// TIA Portal V15.1 export
// export: Created 2024-06-21T08:40:58.1290505Z, ExportSetting WithDefaults, DisplayName Totally Integrated Automation Portal, DisplayVersion V15.1 Update 5, DisplayName TIA Portal Openness, DisplayVersion V15.1 Update 5, DisplayName SINAMICS Startdrive Advanced, DisplayVersion V15.1, DisplayName G130, G150, S120, S150, SINAMICS MV, S210, DisplayVersion V15.1, DisplayName G110M, G120, G120C, G120D, G120P, DisplayVersion V15.1, DisplayName STEP 7 Professional, DisplayVersion V15.1 Update 5, DisplayName STEP 7 Safety, DisplayVersion V15.1, DisplayName WinCC Professional, DisplayVersion V15.1 Update 5, DisplayName SIMATIC Visualization Architect, DisplayVersion V15.1
FUNCTION_BLOCK "LETAFuseCPC20PN"   // FB1406, FBD
TITLE = LETAFuseCPC20PN
{ S7_Optimized_Access := 'TRUE' }
AUTHOR : VCC
FAMILY : AlarmHnd
VERSION : 0.1
// stored: AutoNumber false, IsIECCheckEnabled false, IsRetainMemResEnabled false, MemoryReserve 100, SetENOAutomatically False, UDAEnableTagReadback false
   VAR_INPUT
      I_NewShift { ExternalAccessible := 'False'; ExternalVisible := 'False'; ExternalWritable := 'False'} : Bool;   // NewShift / Morning shift
      I_EnableAlarm { ExternalAccessible := 'False'; ExternalVisible := 'False'; ExternalWritable := 'False'} : Bool := TRUE;   // Enable Alarm from upper level
      C_HWInput { ExternalAccessible := 'False'; ExternalVisible := 'False'; ExternalWritable := 'False'} : HW_IO;   // Slot ID from CPC20PN
      C_Block1_TotalCurrent { ExternalAccessible := 'False'; ExternalVisible := 'False'; ExternalWritable := 'False'} : HW_IO;   // Base Module Slot ID Total Current, 0=not in use.
      C_Block1_StatusControl { ExternalAccessible := 'False'; ExternalVisible := 'False'; ExternalWritable := 'False'} : HW_IO;   // Base Module Slot ID Status / Control, 0=not in use.
      "C_Block1_MeasurementU/I" { ExternalAccessible := 'False'; ExternalVisible := 'False'; ExternalWritable := 'False'} : HW_IO;   // Base Module Slot ID Measurement UI, 0=not in use.
      C_Block2_TotalCurrent { ExternalAccessible := 'False'; ExternalVisible := 'False'; ExternalWritable := 'False'} : HW_IO;   // Extension Module Slot ID Total Current, 0=not in use.
      C_Block2_StatusControl { ExternalAccessible := 'False'; ExternalVisible := 'False'; ExternalWritable := 'False'} : HW_IO;   // Extension Module Slot ID Status / Control, 0=not in use.
      "C_Block2_MeasurementU/I" { ExternalAccessible := 'False'; ExternalVisible := 'False'; ExternalWritable := 'False'} : HW_IO;   // Extension Module Slot ID Measurement UI, 0=not in use.
      C_Config { ExternalAccessible := 'False'; ExternalVisible := 'False'; ExternalWritable := 'False'} : "ETAFuseCPC20PNConfig";   // Config
   END_VAR
   VAR_OUTPUT
      O_AlarmABCondition { ExternalAccessible := 'False'; ExternalVisible := 'False'; ExternalWritable := 'False'} : Bool;   // Alarm AB Condition
      O_AlarmA { ExternalAccessible := 'False'; ExternalVisible := 'False'; ExternalWritable := 'False'} : Bool;   // Alarm A
      O_AlarmB { ExternalAccessible := 'False'; ExternalVisible := 'False'; ExternalWritable := 'False'} : Bool;   // Alarm B
      O_AlarmC { ExternalAccessible := 'False'; ExternalVisible := 'False'; ExternalWritable := 'False'} : Bool;   // Alarm C
      O_AlarmD { ExternalAccessible := 'False'; ExternalVisible := 'False'; ExternalWritable := 'False'} : Bool;   // Alarm D
      H_AlarmDWord { ExternalAccessible := 'False'; ExternalVisible := 'False'; ExternalWritable := 'False'} : DWord;   // HMI Animation
   END_VAR
   VAR_IN_OUT
      IO_ETAFuseData : "ETAFuseData";   // ETA fuse status
      H_HMI : "H_HMI";   // Animation
      H_ETAFuseCPC20PN : "H_ETAFuseCPC20PN";   // Animation
   END_VAR
   VAR
      AC_StatusCPC20_Bit0 { ExternalAccessible := 'False'; ExternalVisible := 'False'; ExternalWritable := 'False'} : Bool;   // No configuration data available
      AC_StatusCPC20_Bit1 { ExternalAccessible := 'False'; ExternalVisible := 'False'; ExternalWritable := 'False'} : Bool;   // Invalid configuration data
      AC_StatusCPC20_Bit4 { ExternalAccessible := 'False'; ExternalVisible := 'False'; ExternalWritable := 'False'} : Bool;   // Command buffer overflow
      AC_StatusCPC20_Bit7 { ExternalAccessible := 'False'; ExternalVisible := 'False'; ExternalWritable := 'False'} : Bool;   // No communication with at least one PWR board
      AC_StatusCPC20_Bit9 { ExternalAccessible := 'False'; ExternalVisible := 'False'; ExternalWritable := 'False'} : Bool;   // CPC tempory error
      AC_StatusCPC20_Bit10 { ExternalAccessible := 'False'; ExternalVisible := 'False'; ExternalWritable := 'False'} : Bool;   // CPC hardware error
      AC_ReadNomCurr { ExternalAccessible := 'False'; ExternalVisible := 'False'; ExternalWritable := 'False'} : Bool;   // Overtime Reading of nominal current
      AlarmABCondition { ExternalAccessible := 'False'; ExternalVisible := 'False'; ExternalWritable := 'False'} : Bool;   // Alarm AB Condition
      AlarmA { ExternalAccessible := 'False'; ExternalVisible := 'False'; ExternalWritable := 'False'} : Bool;   // Alarm A
      AlarmB { ExternalAccessible := 'False'; ExternalVisible := 'False'; ExternalWritable := 'False'} : Bool;   // Alarm B
      AlarmC { ExternalAccessible := 'False'; ExternalVisible := 'False'; ExternalWritable := 'False'} : Bool;   // Alarm C
      AlarmD { ExternalAccessible := 'False'; ExternalVisible := 'False'; ExternalWritable := 'False'} : Bool;   // Alarm D
      ReadNominalCurrentActive { ExternalAccessible := 'False'; ExternalVisible := 'False'; ExternalWritable := 'False'} : Bool;   // Reading of nominal current is active
      EnableAlarm { ExternalAccessible := 'False'; ExternalVisible := 'False'; ExternalWritable := 'False'} : Bool;   // Enable Alarm from upper level
   END_VAR
   VAR RETAIN
      H_ReadNomCurr { ExternalAccessible := 'False'; ExternalVisible := 'False'; ExternalWritable := 'False'} : Bool;   // HMI Command - Read nominal current
      H_CancelReadNomCurr { ExternalAccessible := 'False'; ExternalVisible := 'False'; ExternalWritable := 'False'} : Bool;   // HMI Command - Cancel Read nominal current
   END_VAR
   VAR
      H_UpChannel { ExternalAccessible := 'False'; ExternalVisible := 'False'; ExternalWritable := 'False'} : Bool;   // HMI Command - UP channel selection
      H_DownChannel { ExternalAccessible := 'False'; ExternalVisible := 'False'; ExternalWritable := 'False'} : Bool;   // HMI Command - DOWN channel selection
      H_SwitchON { ExternalAccessible := 'False'; ExternalVisible := 'False'; ExternalWritable := 'False'} : Bool;   // HMICmd / HMI Command - Switch On
      H_SwitchOFF { ExternalAccessible := 'False'; ExternalVisible := 'False'; ExternalWritable := 'False'} : Bool;   // HMICmd / HMI Command - Switch Off
      H_Transfer { ExternalAccessible := 'False'; ExternalVisible := 'False'; ExternalWritable := 'False'} : Bool;   // HMICmd / HMI Command - Transfer
      H_Reset { ExternalAccessible := 'False'; ExternalVisible := 'False'; ExternalWritable := 'False'} : Bool;   // HMICmd / HMI Command - Reset
      _ETAFuseCPC20PNSub { ExternalAccessible := 'False'; ExternalVisible := 'False'; ExternalWritable := 'False'} : "LETAFuseCPC20PNSub";   // FB
   END_VAR
   VAR DB_SPECIFIC
      T_ResetControl { ExternalAccessible := 'False'; ExternalVisible := 'False'; ExternalWritable := 'False'} : TON_TIME;   // Timer
      T_EnableAlarm { ExternalAccessible := 'False'; ExternalVisible := 'False'; ExternalWritable := 'False'} : TON_TIME;   // Timer
   END_VAR
   VAR
      Edge { ExternalAccessible := 'False'; ExternalVisible := 'False'; ExternalWritable := 'False'} : Array[0..10] of Bool;   // Edge
   END_VAR
   VAR_TEMP   // added for the SCL form of the ladder/FBD networks
      _w1 : Bool;
      _w2 : Bool;
   END_VAR
BEGIN

REGION Network 1: **** 1 - Inputs **** Extract The Commands From HMI
   // Extract The Commands From HMI
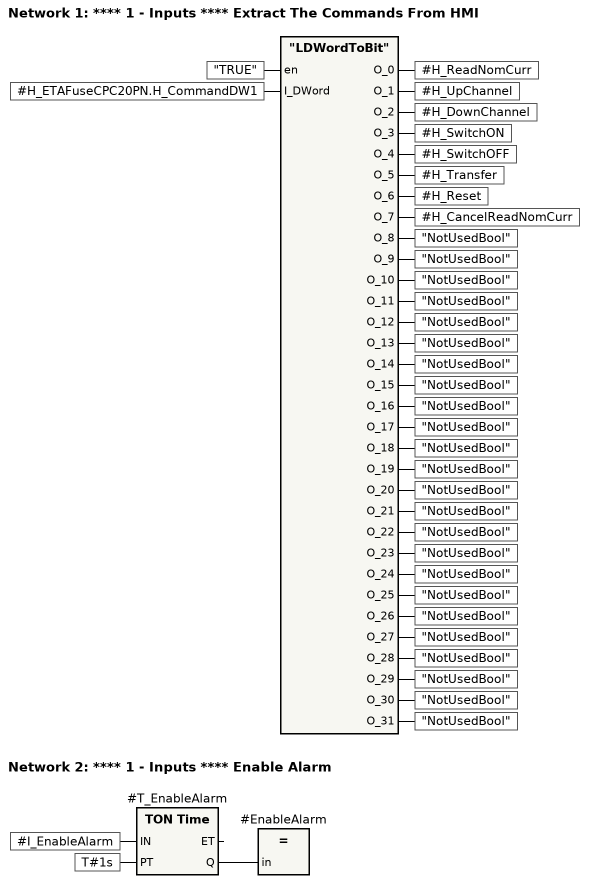
   IF "TRUE" THEN
       "LDWordToBit"(I_DWord := #H_ETAFuseCPC20PN.H_CommandDW1,
                     O_0 => #H_ReadNomCurr,
                     O_1 => #H_UpChannel,
                     O_2 => #H_DownChannel,
                     O_3 => #H_SwitchON,
                     O_4 => #H_SwitchOFF,
                     O_5 => #H_Transfer,
                     O_6 => #H_Reset,
                     O_7 => #H_CancelReadNomCurr,
                     O_8 => "NotUsedBool",
                     O_9 => "NotUsedBool",
                     O_10 => "NotUsedBool",
                     O_11 => "NotUsedBool",
                     O_12 => "NotUsedBool",
                     O_13 => "NotUsedBool",
                     O_14 => "NotUsedBool",
                     O_15 => "NotUsedBool",
                     O_16 => "NotUsedBool",
                     O_17 => "NotUsedBool",
                     O_18 => "NotUsedBool",
                     O_19 => "NotUsedBool",
                     O_20 => "NotUsedBool",
                     O_21 => "NotUsedBool",
                     O_22 => "NotUsedBool",
                     O_23 => "NotUsedBool",
                     O_24 => "NotUsedBool",
                     O_25 => "NotUsedBool",
                     O_26 => "NotUsedBool",
                     O_27 => "NotUsedBool",
                     O_28 => "NotUsedBool",
                     O_29 => "NotUsedBool",
                     O_30 => "NotUsedBool",
                     O_31 => "NotUsedBool");
   END_IF;
END_REGION

REGION Network 2: **** 1 - Inputs **** Enable Alarm
   #T_EnableAlarm(IN := #I_EnableAlarm, PT := T#1s);   // TON
   #EnableAlarm := #T_EnableAlarm.Q;
END_REGION

REGION Network 3: **** 4.3 - Machine status - Operator Selection **** Selected Channel
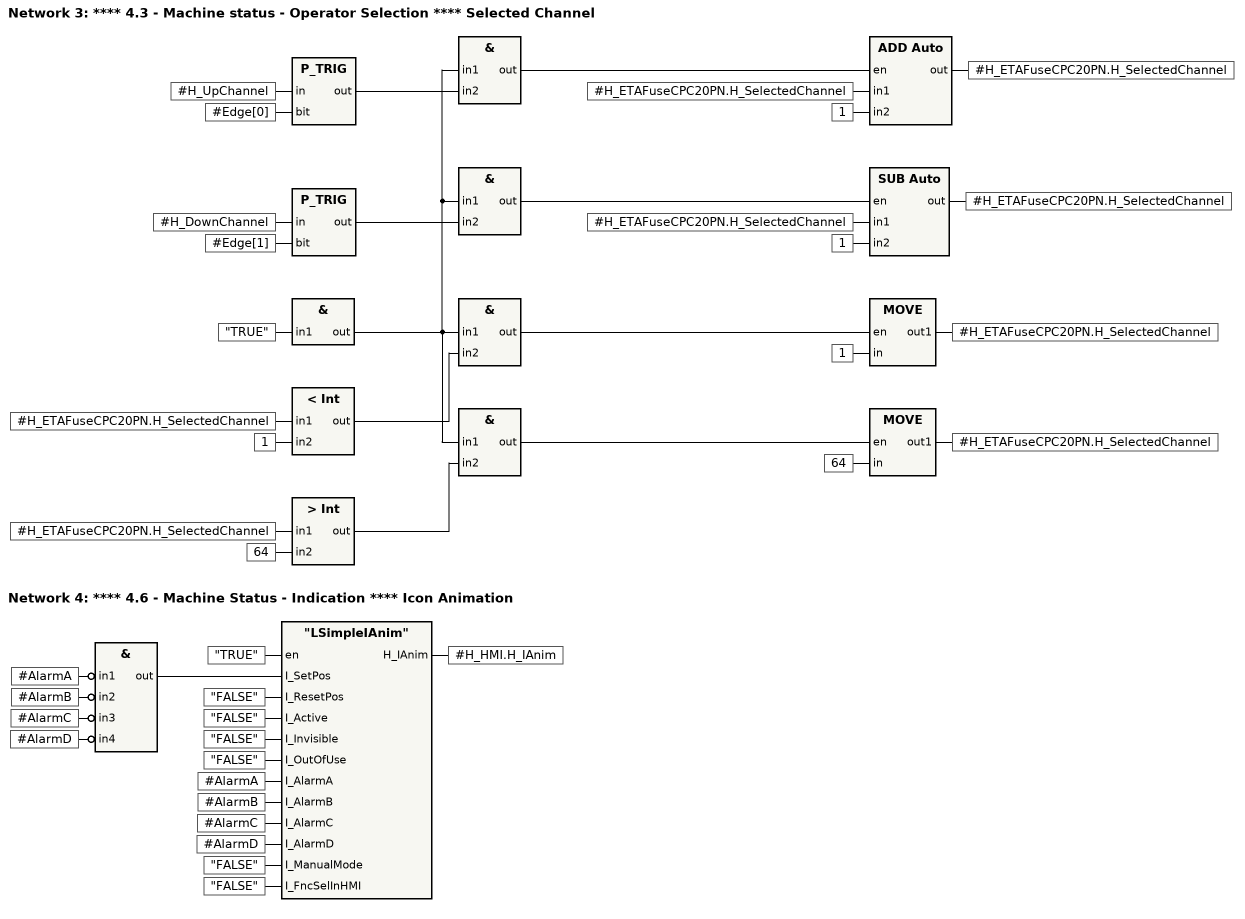
   #_w1 := #H_UpChannel AND NOT #Edge[0];   // rising edge
   #Edge[0] := #H_UpChannel;
   IF "TRUE" AND #_w1 THEN
       #H_ETAFuseCPC20PN.H_SelectedChannel := #H_ETAFuseCPC20PN.H_SelectedChannel + 1;
   END_IF;
   #_w2 := #H_DownChannel AND NOT #Edge[1];   // rising edge
   #Edge[1] := #H_DownChannel;
   IF "TRUE" AND #_w2 THEN
       #H_ETAFuseCPC20PN.H_SelectedChannel := #H_ETAFuseCPC20PN.H_SelectedChannel - 1;
   END_IF;
   IF "TRUE" AND (#H_ETAFuseCPC20PN.H_SelectedChannel < 1) THEN
       #H_ETAFuseCPC20PN.H_SelectedChannel := 1;
   END_IF;
   IF "TRUE" AND (#H_ETAFuseCPC20PN.H_SelectedChannel > 64) THEN
       #H_ETAFuseCPC20PN.H_SelectedChannel := 64;
   END_IF;
END_REGION

REGION Network 4: **** 4.6 - Machine Status - Indication **** Icon Animation
   // Icon Animation
   IF "TRUE" THEN
       "LSimpleIAnim"(I_SetPos := NOT #AlarmA AND NOT #AlarmB AND NOT #AlarmC AND NOT #AlarmD,
                      I_ResetPos := "FALSE",
                      I_Active := "FALSE",
                      I_Invisible := "FALSE",
                      I_OutOfUse := "FALSE",
                      I_AlarmA := #AlarmA,
                      I_AlarmB := #AlarmB,
                      I_AlarmC := #AlarmC,
                      I_AlarmD := #AlarmD,
                      I_ManualMode := "FALSE",
                      I_FncSelInHMI := "FALSE",
                      H_IAnim => #H_HMI.H_IAnim);
   END_IF;
END_REGION

REGION Network 5: **** 4.6 - Machine Status - Indication **** Animation
   // Animation
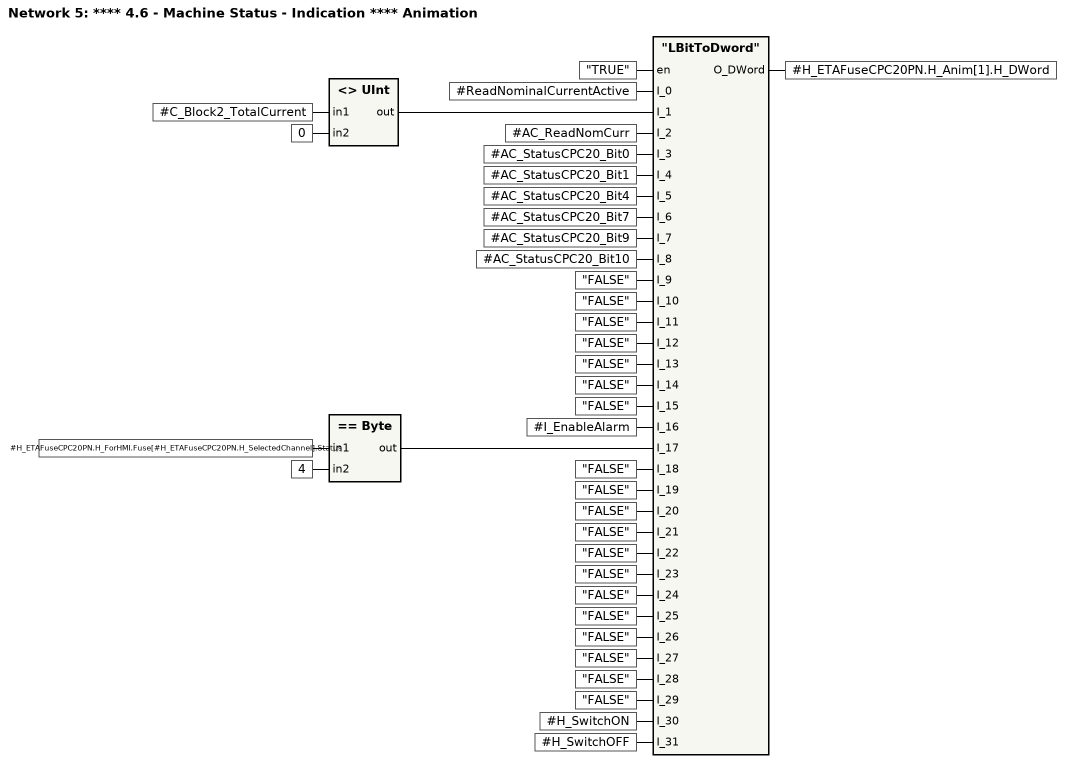
   IF "TRUE" THEN
       "LBitToDword"(I_0 := #ReadNominalCurrentActive,
                     I_1 := #C_Block2_TotalCurrent <> 0,
                     I_2 := #AC_ReadNomCurr,
                     I_3 := #AC_StatusCPC20_Bit0,
                     I_4 := #AC_StatusCPC20_Bit1,
                     I_5 := #AC_StatusCPC20_Bit4,
                     I_6 := #AC_StatusCPC20_Bit7,
                     I_7 := #AC_StatusCPC20_Bit9,
                     I_8 := #AC_StatusCPC20_Bit10,
                     I_9 := "FALSE",
                     I_10 := "FALSE",
                     I_11 := "FALSE",
                     I_12 := "FALSE",
                     I_13 := "FALSE",
                     I_14 := "FALSE",
                     I_15 := "FALSE",
                     I_16 := #I_EnableAlarm,
                     I_17 := #H_ETAFuseCPC20PN.H_ForHMI.Fuse[#H_ETAFuseCPC20PN.H_SelectedChannel].Status = 4,
                     I_18 := "FALSE",
                     I_19 := "FALSE",
                     I_20 := "FALSE",
                     I_21 := "FALSE",
                     I_22 := "FALSE",
                     I_23 := "FALSE",
                     I_24 := "FALSE",
                     I_25 := "FALSE",
                     I_26 := "FALSE",
                     I_27 := "FALSE",
                     I_28 := "FALSE",
                     I_29 := "FALSE",
                     I_30 := #H_SwitchON,
                     I_31 := #H_SwitchOFF,
                     O_DWord => #H_ETAFuseCPC20PN.H_Anim[1].H_DWord);
   END_IF;
END_REGION

REGION Network 6: **** 4.6 - Machine Status - Indication **** Animation
   // Animation
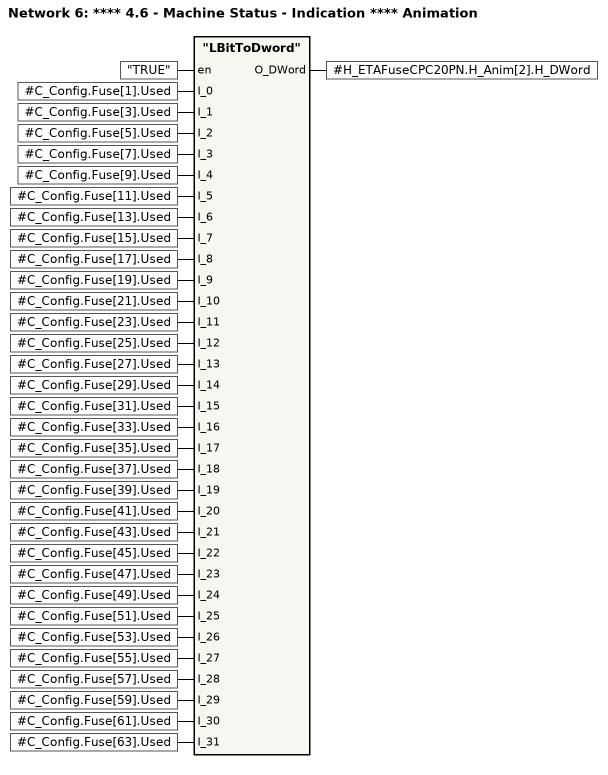
   IF "TRUE" THEN
       "LBitToDword"(I_0 := #C_Config.Fuse[1].Used,
                     I_1 := #C_Config.Fuse[3].Used,
                     I_2 := #C_Config.Fuse[5].Used,
                     I_3 := #C_Config.Fuse[7].Used,
                     I_4 := #C_Config.Fuse[9].Used,
                     I_5 := #C_Config.Fuse[11].Used,
                     I_6 := #C_Config.Fuse[13].Used,
                     I_7 := #C_Config.Fuse[15].Used,
                     I_8 := #C_Config.Fuse[17].Used,
                     I_9 := #C_Config.Fuse[19].Used,
                     I_10 := #C_Config.Fuse[21].Used,
                     I_11 := #C_Config.Fuse[23].Used,
                     I_12 := #C_Config.Fuse[25].Used,
                     I_13 := #C_Config.Fuse[27].Used,
                     I_14 := #C_Config.Fuse[29].Used,
                     I_15 := #C_Config.Fuse[31].Used,
                     I_16 := #C_Config.Fuse[33].Used,
                     I_17 := #C_Config.Fuse[35].Used,
                     I_18 := #C_Config.Fuse[37].Used,
                     I_19 := #C_Config.Fuse[39].Used,
                     I_20 := #C_Config.Fuse[41].Used,
                     I_21 := #C_Config.Fuse[43].Used,
                     I_22 := #C_Config.Fuse[45].Used,
                     I_23 := #C_Config.Fuse[47].Used,
                     I_24 := #C_Config.Fuse[49].Used,
                     I_25 := #C_Config.Fuse[51].Used,
                     I_26 := #C_Config.Fuse[53].Used,
                     I_27 := #C_Config.Fuse[55].Used,
                     I_28 := #C_Config.Fuse[57].Used,
                     I_29 := #C_Config.Fuse[59].Used,
                     I_30 := #C_Config.Fuse[61].Used,
                     I_31 := #C_Config.Fuse[63].Used,
                     O_DWord => #H_ETAFuseCPC20PN.H_Anim[2].H_DWord);
   END_IF;
END_REGION

REGION Network 7: **** 4.6 - Machine Status - Indication **** Animation
   // Animation
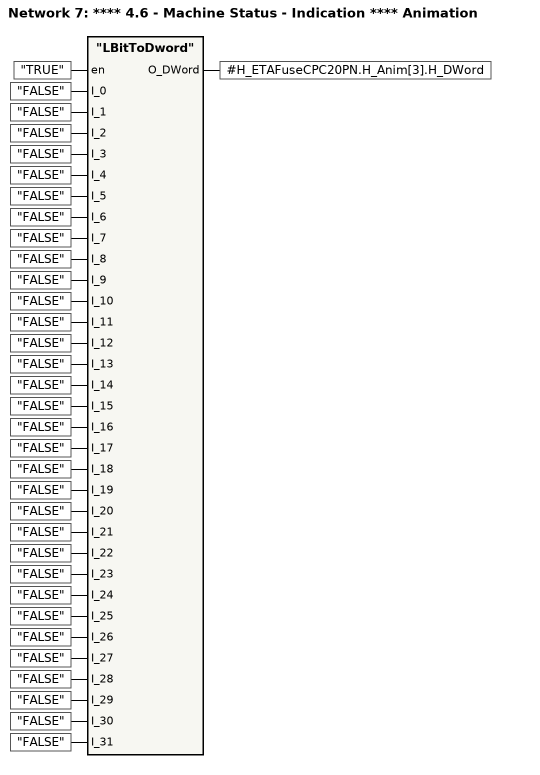
   IF "TRUE" THEN
       "LBitToDword"(I_0 := "FALSE",
                     I_1 := "FALSE",
                     I_2 := "FALSE",
                     I_3 := "FALSE",
                     I_4 := "FALSE",
                     I_5 := "FALSE",
                     I_6 := "FALSE",
                     I_7 := "FALSE",
                     I_8 := "FALSE",
                     I_9 := "FALSE",
                     I_10 := "FALSE",
                     I_11 := "FALSE",
                     I_12 := "FALSE",
                     I_13 := "FALSE",
                     I_14 := "FALSE",
                     I_15 := "FALSE",
                     I_16 := "FALSE",
                     I_17 := "FALSE",
                     I_18 := "FALSE",
                     I_19 := "FALSE",
                     I_20 := "FALSE",
                     I_21 := "FALSE",
                     I_22 := "FALSE",
                     I_23 := "FALSE",
                     I_24 := "FALSE",
                     I_25 := "FALSE",
                     I_26 := "FALSE",
                     I_27 := "FALSE",
                     I_28 := "FALSE",
                     I_29 := "FALSE",
                     I_30 := "FALSE",
                     I_31 := "FALSE",
                     O_DWord => #H_ETAFuseCPC20PN.H_Anim[3].H_DWord);
   END_IF;
END_REGION

REGION Network 8: **** 4.6 - Machine Status - Indication **** Animation
   // Animation
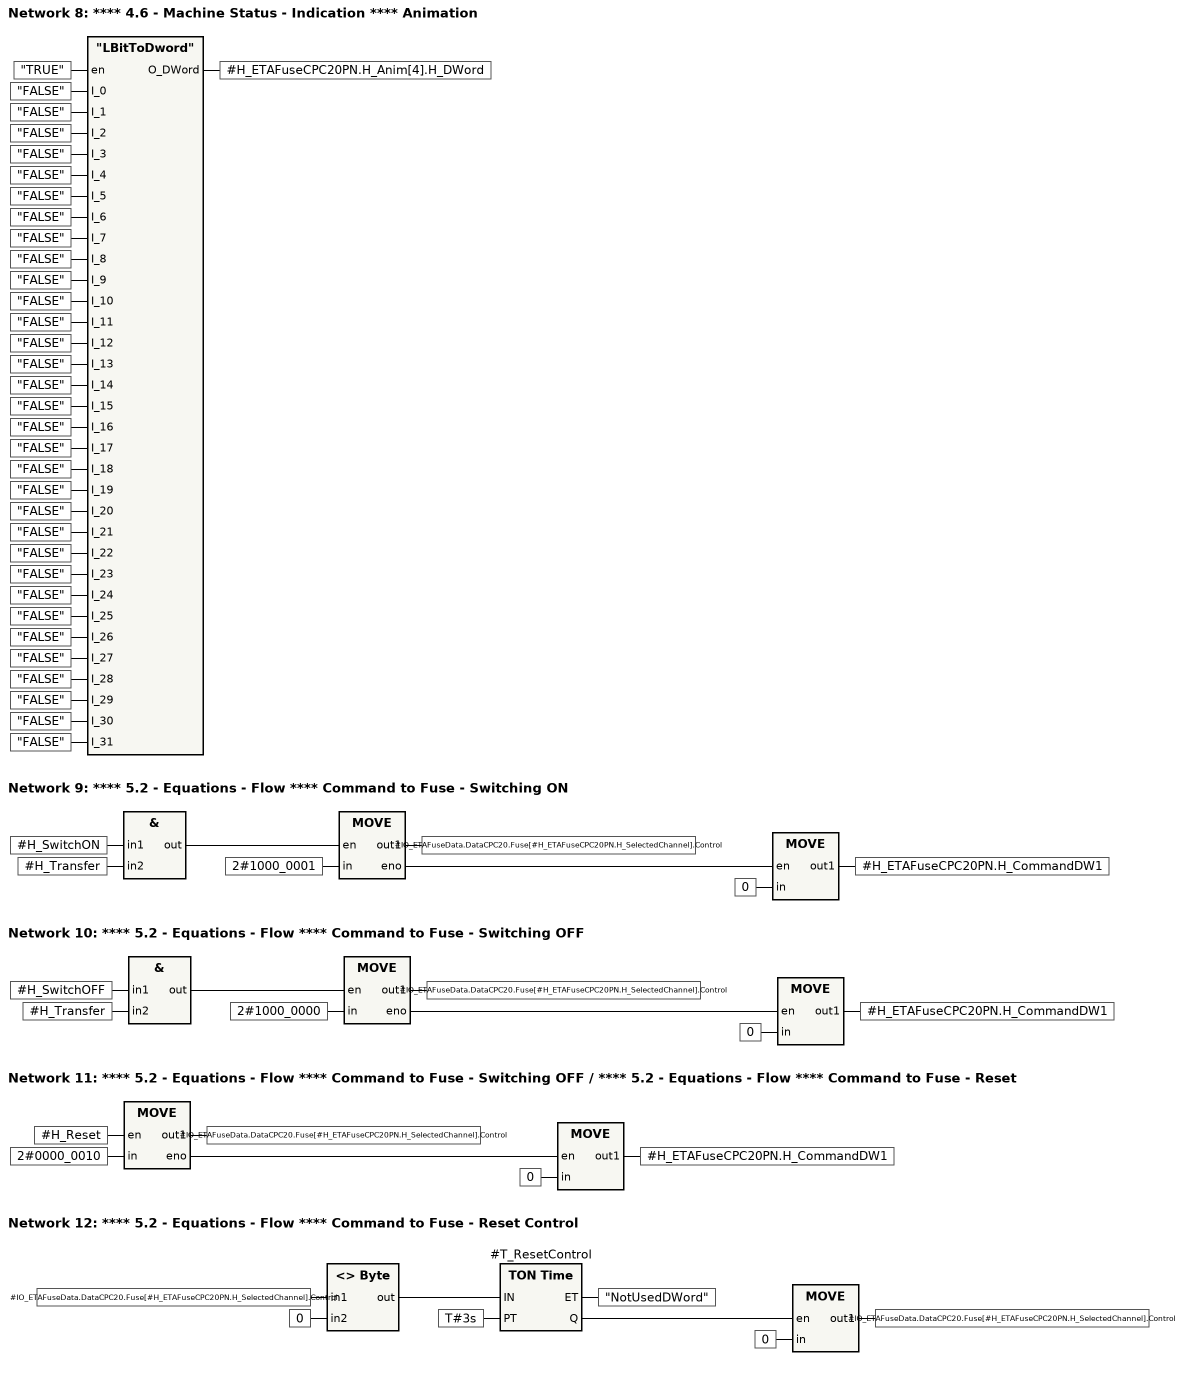
   IF "TRUE" THEN
       "LBitToDword"(I_0 := "FALSE",
                     I_1 := "FALSE",
                     I_2 := "FALSE",
                     I_3 := "FALSE",
                     I_4 := "FALSE",
                     I_5 := "FALSE",
                     I_6 := "FALSE",
                     I_7 := "FALSE",
                     I_8 := "FALSE",
                     I_9 := "FALSE",
                     I_10 := "FALSE",
                     I_11 := "FALSE",
                     I_12 := "FALSE",
                     I_13 := "FALSE",
                     I_14 := "FALSE",
                     I_15 := "FALSE",
                     I_16 := "FALSE",
                     I_17 := "FALSE",
                     I_18 := "FALSE",
                     I_19 := "FALSE",
                     I_20 := "FALSE",
                     I_21 := "FALSE",
                     I_22 := "FALSE",
                     I_23 := "FALSE",
                     I_24 := "FALSE",
                     I_25 := "FALSE",
                     I_26 := "FALSE",
                     I_27 := "FALSE",
                     I_28 := "FALSE",
                     I_29 := "FALSE",
                     I_30 := "FALSE",
                     I_31 := "FALSE",
                     O_DWord => #H_ETAFuseCPC20PN.H_Anim[4].H_DWord);
   END_IF;
END_REGION

REGION Network 9: **** 5.2 - Equations - Flow **** Command to Fuse - Switching ON
   // Switching ON
   // ENO of a box is taken as its EN; it also drops when the box reports an error
   IF #H_SwitchON AND #H_Transfer THEN
       #IO_ETAFuseData.DataCPC20.Fuse[#H_ETAFuseCPC20PN.H_SelectedChannel].Control := 2#1000_0001;
       #H_ETAFuseCPC20PN.H_CommandDW1 := 0;
   END_IF;
END_REGION

REGION Network 10: **** 5.2 - Equations - Flow **** Command to Fuse - Switching OFF
   // Switching OFF
   // ENO of a box is taken as its EN; it also drops when the box reports an error
   IF #H_SwitchOFF AND #H_Transfer THEN
       #IO_ETAFuseData.DataCPC20.Fuse[#H_ETAFuseCPC20PN.H_SelectedChannel].Control := 2#1000_0000;
       #H_ETAFuseCPC20PN.H_CommandDW1 := 0;
   END_IF;
END_REGION

REGION Network 11: **** 5.2 - Equations - Flow **** Command to Fuse - Switching OFF / **** 5.2 - Equations - Flow **** Command to Fuse - Reset
   // Switching OFF / Reset
   // ENO of a box is taken as its EN; it also drops when the box reports an error
   IF #H_Reset THEN
       #IO_ETAFuseData.DataCPC20.Fuse[#H_ETAFuseCPC20PN.H_SelectedChannel].Control := 2#0000_0010;
       #H_ETAFuseCPC20PN.H_CommandDW1 := 0;
   END_IF;
END_REGION

REGION Network 12: **** 5.2 - Equations - Flow **** Command to Fuse - Reset Control
   #T_ResetControl(IN := #IO_ETAFuseData.DataCPC20.Fuse[#H_ETAFuseCPC20PN.H_SelectedChannel].Control <> 0,   // TON
                   PT := T#3s,
                   ET => "NotUsedDWord");
   IF #T_ResetControl.Q THEN
       #IO_ETAFuseData.DataCPC20.Fuse[#H_ETAFuseCPC20PN.H_SelectedChannel].Control := 0;
   END_IF;
END_REGION

REGION Network 13: **** 7.1 - Submodule - Non-Machine **** ETA CPC20 PN
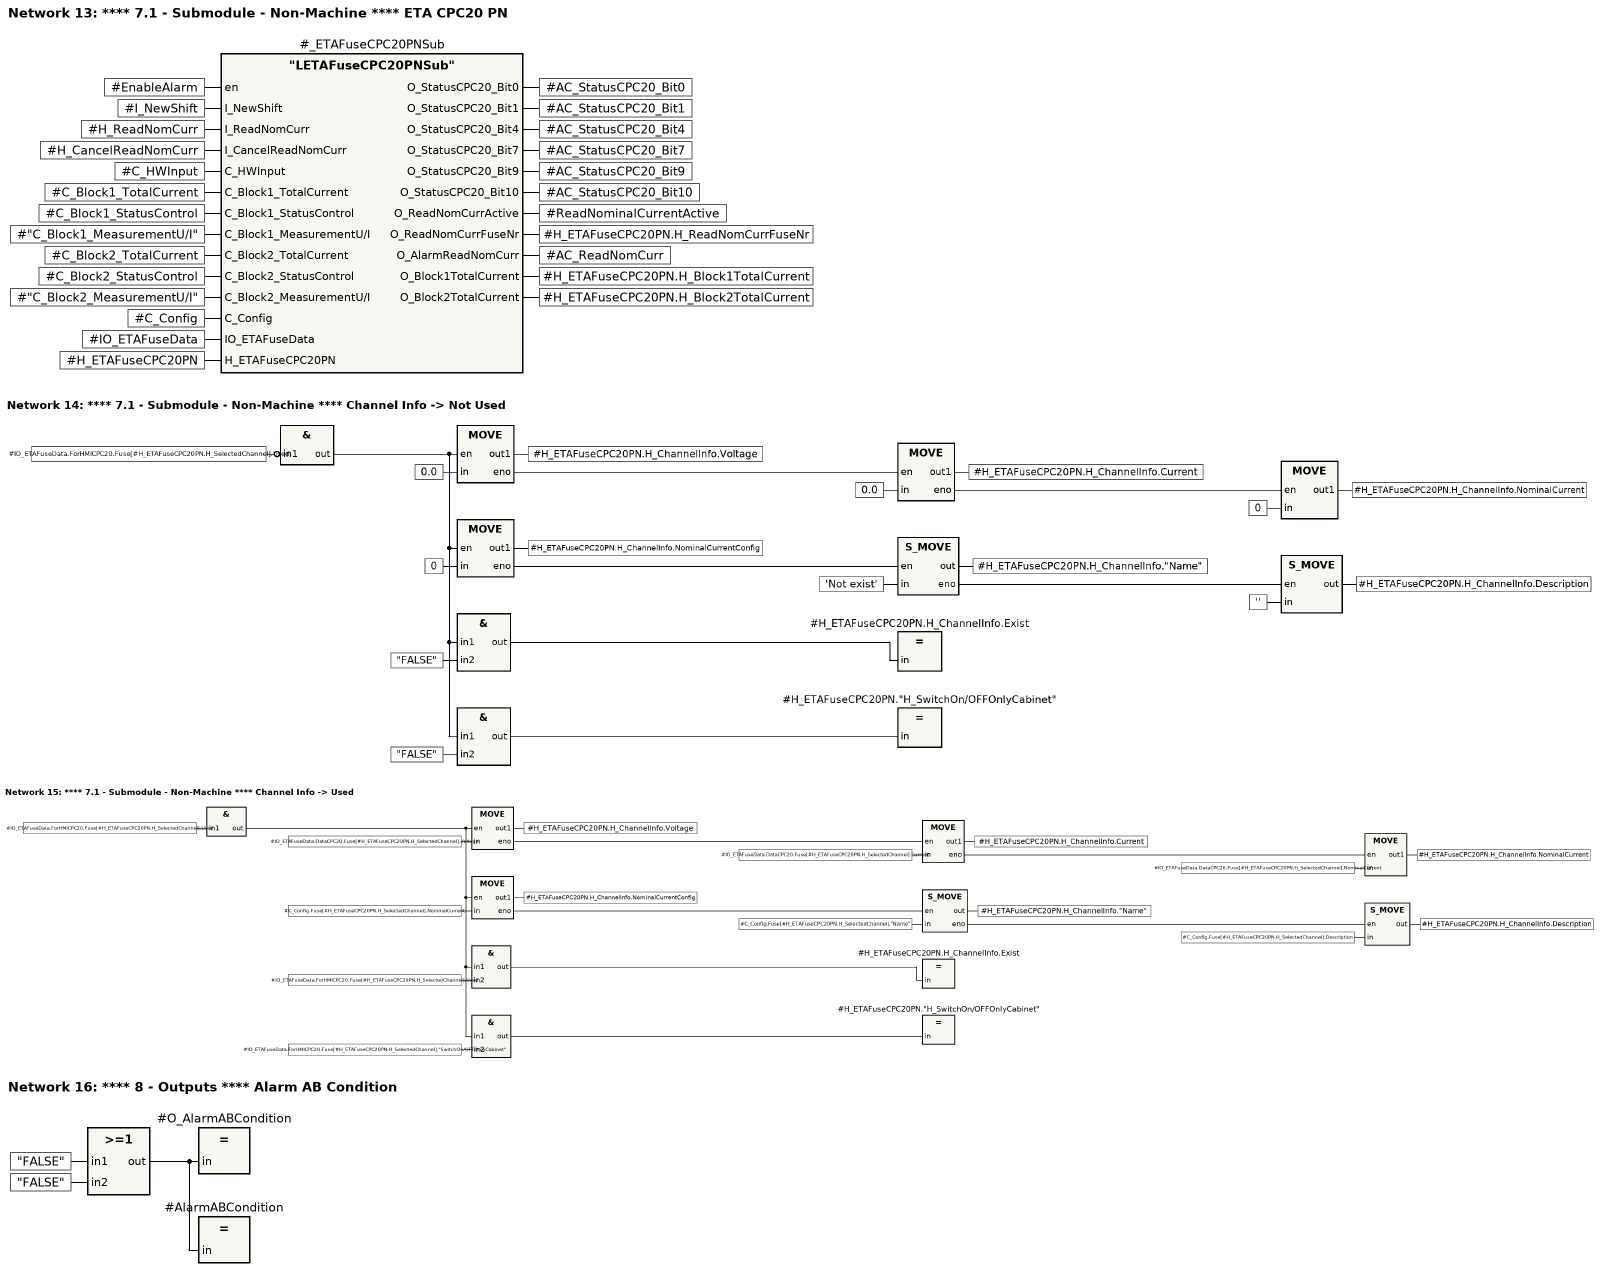
   IF #EnableAlarm THEN
       #_ETAFuseCPC20PNSub(I_NewShift := #I_NewShift,   // "LETAFuseCPC20PNSub"
                           I_ReadNomCurr := #H_ReadNomCurr,
                           I_CancelReadNomCurr := #H_CancelReadNomCurr,
                           C_HWInput := #C_HWInput,
                           C_Block1_TotalCurrent := #C_Block1_TotalCurrent,
                           C_Block1_StatusControl := #C_Block1_StatusControl,
                           "C_Block1_MeasurementU/I" := #"C_Block1_MeasurementU/I",
                           C_Block2_TotalCurrent := #C_Block2_TotalCurrent,
                           C_Block2_StatusControl := #C_Block2_StatusControl,
                           "C_Block2_MeasurementU/I" := #"C_Block2_MeasurementU/I",
                           C_Config := #C_Config,
                           IO_ETAFuseData := #IO_ETAFuseData,
                           H_ETAFuseCPC20PN := #H_ETAFuseCPC20PN,
                           O_StatusCPC20_Bit0 => #AC_StatusCPC20_Bit0,
                           O_StatusCPC20_Bit1 => #AC_StatusCPC20_Bit1,
                           O_StatusCPC20_Bit4 => #AC_StatusCPC20_Bit4,
                           O_StatusCPC20_Bit7 => #AC_StatusCPC20_Bit7,
                           O_StatusCPC20_Bit9 => #AC_StatusCPC20_Bit9,
                           O_StatusCPC20_Bit10 => #AC_StatusCPC20_Bit10,
                           O_ReadNomCurrActive => #ReadNominalCurrentActive,
                           O_ReadNomCurrFuseNr => #H_ETAFuseCPC20PN.H_ReadNomCurrFuseNr,
                           O_AlarmReadNomCurr => #AC_ReadNomCurr,
                           O_Block1TotalCurrent => #H_ETAFuseCPC20PN.H_Block1TotalCurrent,
                           O_Block2TotalCurrent => #H_ETAFuseCPC20PN.H_Block2TotalCurrent);
   END_IF;
END_REGION

REGION Network 14: **** 7.1 - Submodule - Non-Machine **** Channel Info -> Not Used
   #_w1 := NOT #IO_ETAFuseData.ForHMICPC20.Fuse[#H_ETAFuseCPC20PN.H_SelectedChannel].Used;
   IF #_w1 THEN
       #H_ETAFuseCPC20PN.H_ChannelInfo.Voltage := 0.0;
       #H_ETAFuseCPC20PN.H_ChannelInfo.Current := 0.0;
       #H_ETAFuseCPC20PN.H_ChannelInfo.NominalCurrent := 0;
       #H_ETAFuseCPC20PN.H_ChannelInfo.NominalCurrentConfig := 0;
       #H_ETAFuseCPC20PN.H_ChannelInfo."Name" := 'Not exist';
       #H_ETAFuseCPC20PN.H_ChannelInfo.Description := '';
   END_IF;
   #H_ETAFuseCPC20PN.H_ChannelInfo.Exist := #_w1 AND "FALSE";
   #H_ETAFuseCPC20PN."H_SwitchOn/OFFOnlyCabinet" := #_w1 AND "FALSE";
END_REGION

REGION Network 15: **** 7.1 - Submodule - Non-Machine **** Channel Info -> Used
   IF #IO_ETAFuseData.ForHMICPC20.Fuse[#H_ETAFuseCPC20PN.H_SelectedChannel].Used THEN
       #H_ETAFuseCPC20PN.H_ChannelInfo.Voltage := #IO_ETAFuseData.DataCPC20.Fuse[#H_ETAFuseCPC20PN.H_SelectedChannel].Voltage;
       #H_ETAFuseCPC20PN.H_ChannelInfo.Current := #IO_ETAFuseData.DataCPC20.Fuse[#H_ETAFuseCPC20PN.H_SelectedChannel].Current;
       #H_ETAFuseCPC20PN.H_ChannelInfo.NominalCurrent := #IO_ETAFuseData.DataCPC20.Fuse[#H_ETAFuseCPC20PN.H_SelectedChannel].NominalCurrent;
       #H_ETAFuseCPC20PN.H_ChannelInfo.NominalCurrentConfig := #C_Config.Fuse[#H_ETAFuseCPC20PN.H_SelectedChannel].NominalCurrent;
       #H_ETAFuseCPC20PN.H_ChannelInfo."Name" := #C_Config.Fuse[#H_ETAFuseCPC20PN.H_SelectedChannel]."Name";
       #H_ETAFuseCPC20PN.H_ChannelInfo.Description := #C_Config.Fuse[#H_ETAFuseCPC20PN.H_SelectedChannel].Description;
   END_IF;
   #H_ETAFuseCPC20PN.H_ChannelInfo.Exist := #IO_ETAFuseData.ForHMICPC20.Fuse[#H_ETAFuseCPC20PN.H_SelectedChannel].Used AND #IO_ETAFuseData.ForHMICPC20.Fuse[#H_ETAFuseCPC20PN.H_SelectedChannel].Used;
   #H_ETAFuseCPC20PN."H_SwitchOn/OFFOnlyCabinet" := #IO_ETAFuseData.ForHMICPC20.Fuse[#H_ETAFuseCPC20PN.H_SelectedChannel].Used AND #IO_ETAFuseData.ForHMICPC20.Fuse[#H_ETAFuseCPC20PN.H_SelectedChannel]."SwitchOn/OFFOnlyCabinet";
END_REGION

REGION Network 16: **** 8 - Outputs **** Alarm AB Condition
   // Alarm AB Condition
   #O_AlarmABCondition := "FALSE" OR "FALSE";
   #AlarmABCondition := #O_AlarmABCondition;
END_REGION

REGION Network 17: **** 9 - Alarm Summary **** Alarm A
   // Alarm A
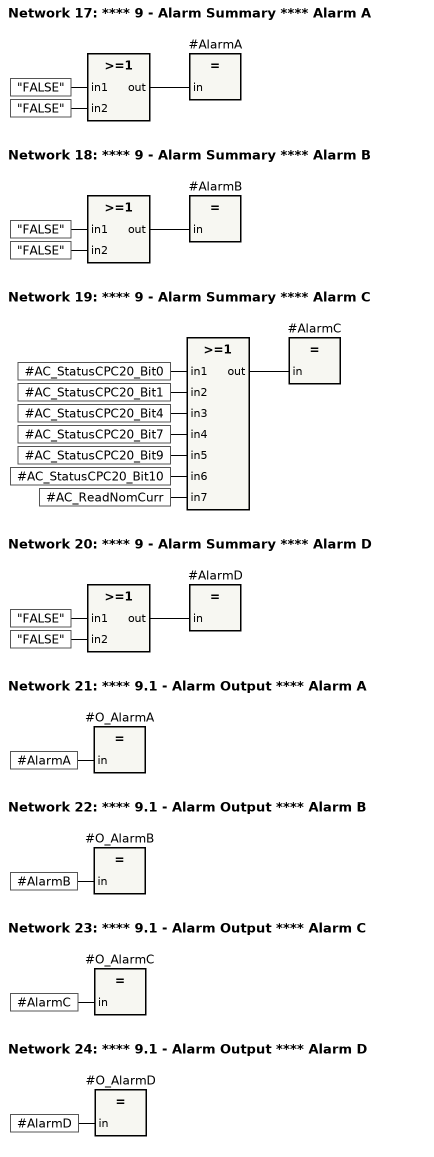
   #AlarmA := "FALSE" OR "FALSE";
END_REGION

REGION Network 18: **** 9 - Alarm Summary **** Alarm B
   // Alarm B
   #AlarmB := "FALSE" OR "FALSE";
END_REGION

REGION Network 19: **** 9 - Alarm Summary **** Alarm C
   // Alarm C
   #AlarmC := #AC_StatusCPC20_Bit0 OR #AC_StatusCPC20_Bit1 OR #AC_StatusCPC20_Bit4 OR #AC_StatusCPC20_Bit7 OR #AC_StatusCPC20_Bit9 OR #AC_StatusCPC20_Bit10 OR #AC_ReadNomCurr;
END_REGION

REGION Network 20: **** 9 - Alarm Summary **** Alarm D
   // Alarm D
   #AlarmD := "FALSE" OR "FALSE";
END_REGION

REGION Network 21: **** 9.1 - Alarm Output **** Alarm A
   // Alarm A
   #O_AlarmA := #AlarmA;
END_REGION

REGION Network 22: **** 9.1 - Alarm Output **** Alarm B
   // Alarm B
   #O_AlarmB := #AlarmB;
END_REGION

REGION Network 23: **** 9.1 - Alarm Output **** Alarm C
   // Alarm C
   #O_AlarmC := #AlarmC;
END_REGION

REGION Network 24: **** 9.1 - Alarm Output **** Alarm D
   // Alarm D
   #O_AlarmD := #AlarmD;
END_REGION

REGION Network 25: **** 9.2 - Alarm DWord**** Alarm To DWord
   // Alarm To Word
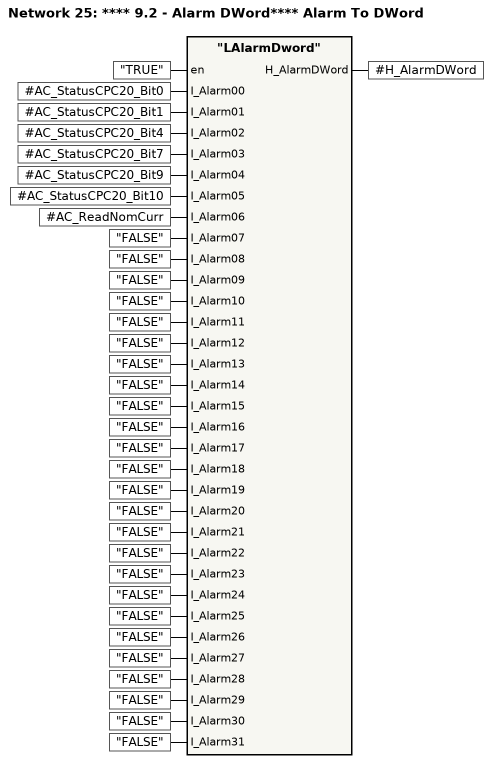
   IF "TRUE" THEN
       "LAlarmDword"(I_Alarm00 := #AC_StatusCPC20_Bit0,
                     I_Alarm01 := #AC_StatusCPC20_Bit1,
                     I_Alarm02 := #AC_StatusCPC20_Bit4,
                     I_Alarm03 := #AC_StatusCPC20_Bit7,
                     I_Alarm04 := #AC_StatusCPC20_Bit9,
                     I_Alarm05 := #AC_StatusCPC20_Bit10,
                     I_Alarm06 := #AC_ReadNomCurr,
                     I_Alarm07 := "FALSE",
                     I_Alarm08 := "FALSE",
                     I_Alarm09 := "FALSE",
                     I_Alarm10 := "FALSE",
                     I_Alarm11 := "FALSE",
                     I_Alarm12 := "FALSE",
                     I_Alarm13 := "FALSE",
                     I_Alarm14 := "FALSE",
                     I_Alarm15 := "FALSE",
                     I_Alarm16 := "FALSE",
                     I_Alarm17 := "FALSE",
                     I_Alarm18 := "FALSE",
                     I_Alarm19 := "FALSE",
                     I_Alarm20 := "FALSE",
                     I_Alarm21 := "FALSE",
                     I_Alarm22 := "FALSE",
                     I_Alarm23 := "FALSE",
                     I_Alarm24 := "FALSE",
                     I_Alarm25 := "FALSE",
                     I_Alarm26 := "FALSE",
                     I_Alarm27 := "FALSE",
                     I_Alarm28 := "FALSE",
                     I_Alarm29 := "FALSE",
                     I_Alarm30 := "FALSE",
                     I_Alarm31 := "FALSE",
                     H_AlarmDWord => #H_AlarmDWord);
   END_IF;
END_REGION
END_FUNCTION_BLOCK
